// TIA Portal V20 export
DATA_BLOCK "Sensor"   // DB198
{ S7_Optimized_Access := 'TRUE' }
// stored: MemoryReserve 100
   VAR
      EM3 : Array[0..2] of Bool;
      EM4 : Array[0..23] of Bool;
      EM5 : Array[0..23] of Bool;
      EM6 : Array[0..38] of Bool;
      EM7 : Array[0..24] of Bool;
   END_VAR
BEGIN
   // EM3[0] : COMPENSATOR LIMIT SENSOR(-)
   // EM3[1] : COMPENSATOR LIMIT SENSOR(+)
   // EM3[2] : COMPENSATOR HOME SENSOR
   // EM4[0] : ANODE MAIN P&P1 X-AXIS LIMITS SENSOR(-)
   // EM4[1] : ANODE MAIN P&P1 X-AXIS LIMITS SENSOR(+)
   // EM4[2] : ANODE MAIN P&P2 LIMITS SENSOR(-)
   // EM4[3] : ANODE MAIN P&P2 LIMITS SENSOR(+)
   // EM4[4] : ANODE MAIN P&P1 X-AXIS LIMITS SENSOR HOME
   // EM4[5] : ANODE MAIN P&P2 LIMITS SENSOR HOME
   // EM4[6] : ANODE MAIN P&P1 Z-AXIS LIMIT SENSOR(-)
   // EM4[7] : ANODE MAIN P&P1 Z-AXIS LIMIT SENSOR(+)
   // EM4[8] : ANODE MAIN P&P1 Y-AXIS LIMIT SENSOR(-)
   // EM4[9] : ANODE MAIN P&P1 Y-AXIS LIMIT SENSOR(+)
   // EM4[10] : ANODE MAIN P&P1 Z-AXIS HOME SENSOR
   // EM4[11] : ANODE MAIN P&P1 Y-AXIS HOME SENSOR
   // EM4[12] : ANODE MAIN P&P2 Z-AXIS LIMIT SENSOR(-)
   // EM4[13] : ANODE MAIN P&P2 Z-AXIS HOME SENSOR
   // EM4[14] : ANODE MAIN P&P2 Z-AXIS LIMIT SENSOR(+)
   // EM4[15] : ANODE ALIGN TABLE X-AXIS LIMIT SENSOR(-)
   // EM4[16] : ANODE ALIGN TABLE X-AXIS LIMIT SENSOR(+)
   // EM4[17] : ANODE ALIGN TABLE Y1-AXIS LIMIT SENSOR(-)
   // EM4[18] : ANODE ALIGN TABLE Y1-AXIS LIMIT SENSOR(+)
   // EM4[19] : ANODE ALIGN TABLE Y2-AXIS LIMIT SENSOR(-)
   // EM4[20] : ANODE ALIGN TABLE Y2-AXIS LIMIT SENSOR(+)
   // EM4[21] : ANODE ALIGN TABLE X-AXIS HOME SENSOR
   // EM4[22] : ANODE ALIGN TABLE Y1-AXIS HOME SENSOR
   // EM4[23] : ANODE ALIGN TABLE Y2-AXIS HOME SENSOR
   // EM5[0] : CATHODE MAIN P&P1 X-AXIS LIMITS SENSOR(-)
   // EM5[1] : CATHODE MAIN P&P1 X-AXIS LIMITS SENSOR(+)
   // EM5[2] : CATHODE MAIN P&P2 X-AXIS LIMITS SENSOR(-)
   // EM5[3] : CATHODE MAIN P&P2 X-AXIS LIMITS SENSOR(+)
   // EM5[4] : CATHODE MAIN P&P1 X-AXIS LIMITS SENSOR HOME
   // EM5[5] : CATHODE MAIN P&P2 X-AXIS LIMITS SENSOR HOME
   // EM5[6] : CATHODE MAIN P&P1 Z-AXIS LIMIT SENSOR(-)
   // EM5[7] : CATHODE MAIN P&P1 Z-AXIS LIMIT SENSOR(+)
   // EM5[8] : CATHODE MAIN P&P1 Y-AXIS LIMIT SENSOR(-)
   // EM5[9] : CATHODE MAIN P&P1 Y-AXIS LIMIT SENSOR(+)
   // EM5[10] : CATHODE MAIN P&P1 Z-AXIS HOME SENSOR
   // EM5[11] : CATHODE MAIN P&P1 Y-AXIS HOME SENSOR
   // EM5[12] : CATHODE MAIN P&P2 Z-AXIS LIMIT SENSOR(-)
   // EM5[13] : CATHODE MAIN P&P2 Z-AXIS HOME SENSOR
   // EM5[14] : CATHODE MAIN P&P2 Z-AXIS LIMIT SENSOR(+)
   // EM5[15] : CATHODE ALIGN TABLE X-AXIS LIMIT SENSOR(-)
   // EM5[16] : CATHODE ALIGN TABLE X-AXIS LIMIT SENSOR(+)
   // EM5[17] : CATHODE ALIGN TABLE Y1-AXIS LIMIT SENSOR(-)
   // EM5[18] : CATHODE ALIGN TABLE Y1-AXIS LIMIT SENSOR(+)
   // EM5[19] : CATHODE ALIGN TABLE Y2-AXIS LIMIT SENSOR(-)
   // EM5[20] : CATHODE ALIGN TABLE Y2-AXIS LIMIT SENSOR(+)
   // EM5[21] : CATHODE ALIGN TABLE X-AXIS HOME SENSOR
   // EM5[22] : CATHODE ALIGN TABLE Y1-AXIS HOME SENSOR
   // EM5[23] : CATHODE ALIGN TABLE Y2-AXIS HOME SENSOR
   // EM6[0] : FINAL ROLLER FRONT LIMIT SENSOR(-)
   // EM6[1] : FINAL ROLLER FRONT HOME SENSOR
   // EM6[2] : FINAL ROLLER FRONT LIMIT SENSOR(+)
   // EM6[3] : FINAL ROLLER REAR LIMIT SENSOR(-)
   // EM6[4] : FINAL ROLLER REAR HOME SENSOR
   // EM6[5] : FINAL ROLLER REAR LIMIT SENSOR(+)
   // EM6[6] : ANODE MANDREL REAR Y AXIS LIMIT SENSOR(-)
   // EM6[7] : ANODE MANDREL REAR Y AXIS LIMIT SENSOR(+)
   // EM6[8] : ANODE MANDREL REAR Z AXIS LIMIT SENSOR(-)
   // EM6[9] : ANODE MANDREL REAR Z AXIS LIMIT SENSOR(+)
   // EM6[10] : ANODE MANDREL FRONT Y AXIS LIMIT SENSOR(-)
   // EM6[11] : ANODE MANDREL FRONT Y AXIS LIMIT SENSOR(+)
   // EM6[12] : ANODE MANDREL FRONT Z AXIS LIMIT SENSOR(-)
   // EM6[13] : ANODE MANDREL FRONT Z AXIS LIMIT SENSOR(+)
   // EM6[14] : ANODE MANDREL REAR Y AXIS HOME SENSOR
   // EM6[15] : ANODE MANDREL REAR Z AXIS HOME SENSOR
   // EM6[16] : ANODE MANDREL FRONT Y AXIS HOME SENSOR
   // EM6[17] : ANODE MANDREL FRONT Z AXIS HOME SENSOR
   // EM6[18] : CATHODE MANDREL REAR Y AXIS LIMIT SENSOR(-)
   // EM6[19] : CATHODE MANDREL REAR Y AXIS LIMIT SENSOR(+)
   // EM6[20] : CATHODE MANDREL REAR Z AXIS LIMIT SENSOR(-)
   // EM6[21] : CATHODE MANDREL REAR Z AXIS LIMIT SENSOR(+)
   // EM6[22] : CATHODE MANDREL FRONT Y AXIS LIMIT SENSOR(-)
   // EM6[23] : CATHODE MANDREL FRONT Y AXIS LIMIT SENSOR(+)
   // EM6[24] : CATHODE MANDREL FRONT Z AXIS LIMIT SENSOR(-)
   // EM6[25] : CATHODE MANDREL FRONT Z AXIS LIMIT SENSOR(+)
   // EM6[26] : CATHODE MANDREL REAR Y AXIS HOME SENSOR
   // EM6[27] : CATHODE MANDREL REAR Z AXIS HOME SENSOR
   // EM6[28] : CATHODE MANDREL FRONT Y AXIS HOME SENSOR
   // EM6[29] : CATHODE MANDREL FRONT Z AXIS HOME SENSOR
   // EM6[30] : STACK TABLE Z-AXIS LIMIT SENSOR(-)
   // EM6[31] : STACK TABLE Z-AXIS LIMIT SENSOR(+)
   // EM6[32] : STACK TABLE OUT FRONT Z-AXIS LIMIT SENSOR(-)
   // EM6[33] : STACK TABLE OUT FRONT Z-AXIS LIMIT SENSOR(+)
   // EM6[34] : STACK TABLE Z-AXIS HOME SENSOR
   // EM6[35] : STACK TABLE OUT FRONT Z-AXIS HOME SENSOR
   // EM6[36] : STACK TABLE OUT REAR Z-AXIS LIMIT SENSOR(-)
   // EM6[37] : STACK TABLE OUT REAR Z-AXIS LIMIT SENSOR(+)
   // EM6[38] : STACK TABLE OUT REAR Z-AXIS HOME SENSOR
   // EM7[0] : SEPA CLAMP&CUTTER X-AXIS LIMIT SENSOR(-)
   // EM7[1] : SEPA CLAMP&CUTTER X-AXIS HOME SENSOR
   // EM7[2] : SEPA CLAMP&CUTTER X-AXIS LIMIT SENSOR(+)
   // EM7[3] : SEPA GRIPPER X-AXIS LIMIT SENSOR(-)
   // EM7[4] : SEPA GRIPPER X-AXIS HOME SENSOR
   // EM7[5] : SEPA GRIPPER X-AXIS LIMIT SENSOR(+)
   // EM7[6] : SEPA GRIPPER C-AXIS LIMIT SENSOR(+)
   // EM7[7] : SEPA GRIPPER Z-AXIS LIMIT SENSOR(-)
   // EM7[8] : SEPA GRIPPER Z-AXIS LIMIT SENSOR(+)
   // EM7[9] : SEPA GRIPPER Z-AXIS HOME SENSOR
   // EM7[10] : SEPA CLAMP&CUTTER Z-AXIS LIMIT SENSOR(-)
   // EM7[11] : SEPA CLAMP&CUTTER Z-AXIS LIMIT SENSOR(+)
   // EM7[12] : CLAMP&CUTTER Z-AXIS HOME SENSOR
   // EM7[13] : JR WINDER REAR Y-AXIS LIMIT SENSOR(-)
   // EM7[14] : JR WINDER REAR Y-AXIS HOME SENSOR
   // EM7[15] : JR WINDER REAR Y-AXIS LIMIT SENSOR(+)
   // EM7[16] : JR WINDER FRONT Y-AXIS LIMIT SENSOR(-)
   // EM7[17] : JR WINDER FRONT Y-AXIS HOME SENSOR
   // EM7[18] : JR WINDER B-AXIS HOME SENSOR
   // EM7[19] : JR WINDER FRONT Y-AXIS LIMIT SENSOR(+)
   // EM7[20] : SEPA GRIPPER C-AXIS LIMIT SENSOR(-)
   // EM7[21] : PUSHER ROLLER Z-AXIS LIMIT SENSOR(-)
   // EM7[22] : PUSHER ROLLER Z-AXIS HOME SENSOR
   // EM7[23] : PUSHER ROLLER Z-AXIS LIMIT SENSOR(+)
   // EM7[24] : SEPA GRIPPER C-AXIS HOME SENSOR
END_DATA_BLOCK
